// TIA Portal project "2017.10.18_视觉分拣" (V17)

(* hardware
DEVICE "S7-1200 station_1"  S7-1200 Station
   slot 0: "Rack_0"  S7-1200 Rack  Rack  V1.0
   slot 1: "PLC_1"  CPU 1214C DC/DC/Rly  6ES7 214-1HG40-0XB0  V4.5
*)

// ===== PLC "PLC_1"  CPU 1214C DC/DC/Rly =====

VAR_GLOBAL   // PLC tag table "默认变量表"
   "Tag_1" AT %I1.1 : Bool;
   "Tag_2" AT %I1.2 : Bool;
   "Tag_3" AT %MW11 : Int;
   "Tag_4" AT %M7.1 : Bool;
END_VAR

DATA_BLOCK "队列"   // DB1
{ S7_Optimized_Access := 'FALSE' }
VERSION : 0.1
   VAR
      加入队列 : Bool;
      踢出队列 : Bool;
      上一个RLO值2 : Bool;
      上一个RLO值3 : Bool;
      随机生成数据 : Bool;
      上一个RLO值 : Bool;
      时间和日期 : DTL;
      RET_VAL : Int;
      队列数据 : Array[1..10] of UDInt;
      待加入队列的值 : UDInt;
      INDEX : DInt;
      数据缓存 : Array[1..10] of UDInt;
      踢出的数据 : UDInt;
   END_VAR
BEGIN
END_DATA_BLOCK

DATA_BLOCK "队列2_DB_1"   // DB3
{ S7_Optimized_Access := 'TRUE' }
VERSION : 0.1
// stored: InstanceOfName 队列2
"队列2"
BEGIN
END_DATA_BLOCK

FUNCTION_BLOCK "队列2"   // FB1, LAD
{ S7_Optimized_Access := 'TRUE' }
VERSION : 0.1
   VAR_INPUT
      启动 : Bool;
      停止 : Bool;
   END_VAR
   VAR_OUTPUT
      输出 : Bool;
      运行标志位 : Bool;
   END_VAR
   VAR_IN_OUT
      程序步 : Int;
   END_VAR
   VAR
      上一个RLO值1 : Bool;
   END_VAR
   VAR_TEMP
      运行标志位_1 : Bool;
   END_VAR
   VAR CONSTANT
      "a" : Int := 20;
   END_VAR
BEGIN

REGION Network 1
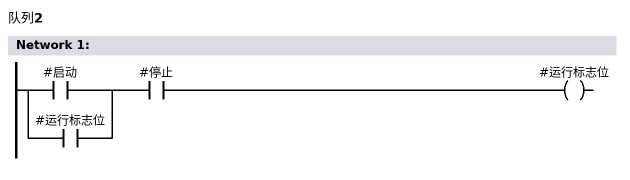
   RUNG wire#powerrail
      Contact( #启动 )
      wire#w1
      Contact( #停止 )
      Coil( #运行标志位 )
   END_RUNG
   RUNG wire#powerrail
      Contact( #运行标志位 )
   END_RUNG wire#w1
   // the same network as SCL:
   #运行标志位 := (#启动 OR #运行标志位) AND #停止;
END_REGION
END_FUNCTION_BLOCK

ORGANIZATION_BLOCK "Main"   // OB1, LAD, ProgramCycle
TITLE = "Main Program Sweep (Cycle)"
{ S7_Optimized_Access := 'TRUE' }
VERSION : 0.1
   VAR_INPUT
      Initial_Call : Bool;   // Initial call of this OB
      Remanence : Bool;   // =True, if remanent data are available
   END_VAR
   VAR_TEMP   // added for the SCL form of the ladder/FBD networks
      _w1 : Bool;
   END_VAR
BEGIN

REGION Network 1: 随机生成数据
   // 上升沿触发 选取DB块中数据           扩张指令里的时钟功能       提取纳秒 类型与纳秒类型一样
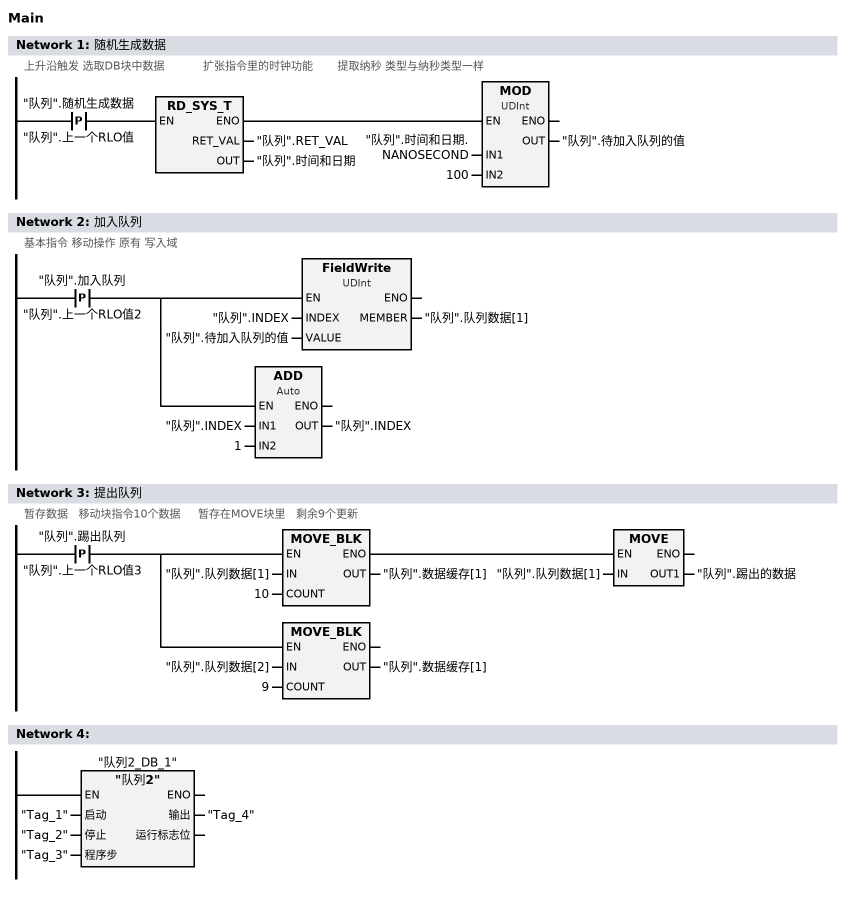
   // ENO of a box is taken as its EN; it also drops when the box reports an error
   #_w1 := "队列".随机生成数据 AND NOT "队列".上一个RLO值;   // rising edge of "队列".随机生成数据
   "队列".上一个RLO值 := "队列".随机生成数据;
   IF #_w1 THEN
       "队列".RET_VAL := RD_SYS_T(OUT => "队列".时间和日期);
       "队列".待加入队列的值 := "队列".时间和日期.NANOSECOND MOD 100;
   END_IF;
END_REGION

REGION Network 2: 加入队列
   // 基本指令 移动操作 原有 写入域
   // no SCL statement known for FieldWrite: written as a call
   #_w1 := "队列".加入队列 AND NOT "队列".上一个RLO值2;   // rising edge of "队列".加入队列
   "队列".上一个RLO值2 := "队列".加入队列;
   IF #_w1 THEN
       FieldWrite(index := "队列".INDEX, value := "队列".待加入队列的值, member => "队列".队列数据[1]);
       "队列".INDEX := "队列".INDEX + 1;
   END_IF;
END_REGION

REGION Network 3: 提出队列
   // 暂存数据   移动块指令10个数据     暂存在MOVE块里   剩余9个更新
   #_w1 := "队列".踢出队列 AND NOT "队列".上一个RLO值3;   // rising edge of "队列".踢出队列
   "队列".上一个RLO值3 := "队列".踢出队列;
   IF #_w1 THEN
       MOVE_BLK(IN := "队列".队列数据[1], COUNT := 10, OUT => "队列".数据缓存[1]);
       "队列".踢出的数据 := "队列".队列数据[1];
       MOVE_BLK(IN := "队列".队列数据[2], COUNT := 9, OUT => "队列".数据缓存[1]);
   END_IF;
END_REGION

REGION Network 4
   RUNG wire#powerrail
      "队列2_DB_1"(启动 := "Tag_1", 停止 := "Tag_2", 程序步 := "Tag_3", 输出 => "Tag_4", 运行标志位 =>)
   END_RUNG
   // the same network as SCL:
   "队列2_DB_1"(启动 := "Tag_1", 停止 := "Tag_2", 程序步 := "Tag_3", 输出 => "Tag_4");   // "队列2"
END_REGION
END_ORGANIZATION_BLOCK